RoboDK station: ESTACION KR10.rdk

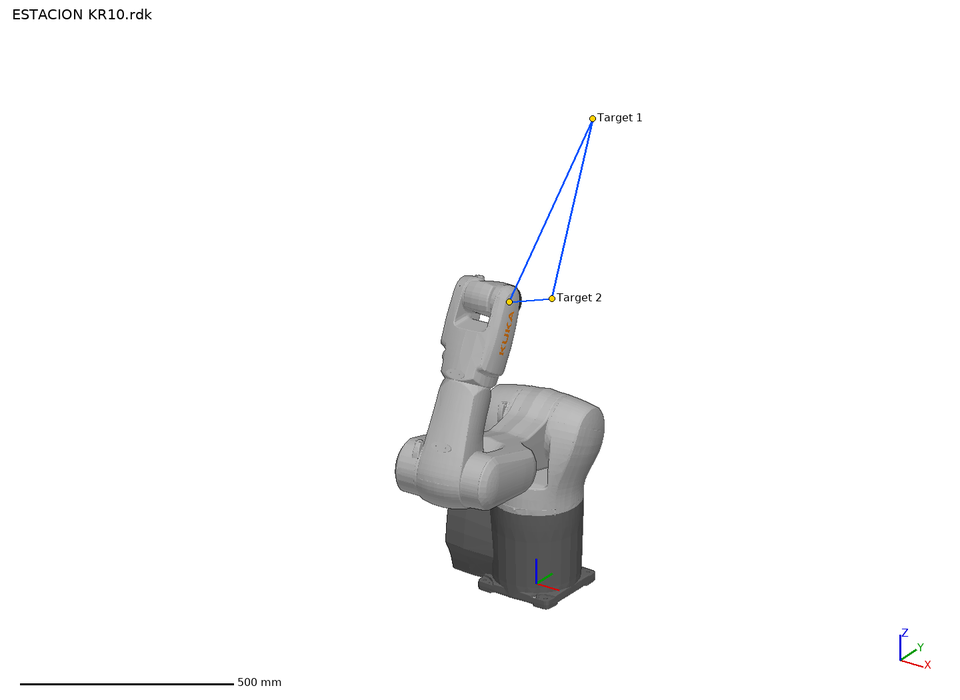
[picture v0: the station drawn from its stored meshes, robots at their saved joint values, targets as dots, program paths as lines]
Station ESTACION KR10 (saved by RoboDK 5.6.7). Poses are relative to the parent item; angles as X-Y-Z fixed-axis rotations.
  - frame KUKA KR 10 R900-2 Base at (0, 0, 0) mm
    - robot KUKA KR 10 R900-2: 6 axes, payload 10 kg, reach 901 mm, repeatability 0.03 mm, weight 52 kg
        modified DH rows (alpha deg, a mm, theta deg, d mm): 0, 0, 0, 400; -90, 25, 0, 0; 0, 455, -90, 0; -90, 25, 0, 420; 90, 0, 0, 0; -90, 0, 180, 90
        joint limits [-170, -190, -120, -185, -120, -350] to [170, 45, 156, 185, 120, 350]; home [0, -90, 90, 0, 0, 0]; saved at [-96.71, -171.34, 110.55, 9.97, 88.38, 69.15]
    - target Target 1 (Cartesian target) at (176.61, -22.09, 1268.28) mm, rotated rx 0 ry 16.57 rz -7.13 deg; joints [7.13, -104.931, 53.874, 0, -22.373, 0] of KUKA KR 10 R900-2
    - target Target 2 (Cartesian target) at (162.12, -169.54, 854.79) mm, rotated rx 176.4 ry 73.21 rz 172.77 deg; joints [65.15, -123.65, 113.03, -66.47, 66.83, 69.15] of KUKA KR 10 R900-2
    - target Target 3 (Cartesian target) at (34.52, -160.15, 806.28) mm, rotated rx -117.97 ry 13.68 rz -11.66 deg; joints [-96.71, -171.34, 110.55, 9.97, 88.38, 69.15] of KUKA KR 10 R900-2
  - program Prog1 (9 instructions, listed below)
  - Python program HandTrackingModule (listed below)
  - Python program FaceHandDetect (listed below)
  - Python program Prog2_vision (listed below)
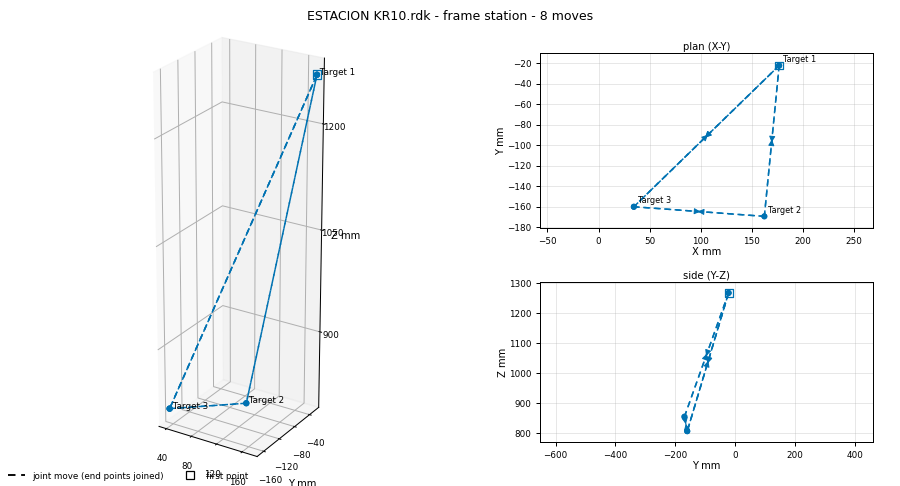
[picture p0: tool path of ESTACION KR10.rdk in frame station, 8 of 8 moves have a stored position in this frame; points joined in program order, loops and branches not executed]

--- program Prog1 (robot KUKA KR 10 R900-2) ---
  Est. Ref.: KUKA KR 10 R900-2 Base
  MoveJ (Target 1)
  MoveJ (Target 2)
  MoveJ (Target 3)
  MoveJ (Target 1)
  MoveJ (Target 3)
  MoveJ (Target 2)
  MoveJ (Target 1)
  MoveJ (Target 3)

--- Python program HandTrackingModule ---
import cv2 as cv
import mediapipe as mp
import time
import math
import numpy as np
import matplotlib.pyplot as plt

## EN PROGRESSO ###

class handDetector():
    def __init__(self,mode=False, maxHands=2,modelC=1,detectConf=0.5,trackConf=0.5):
        self.mode=mode
        self.maxHands=maxHands
        self.modelC = modelC
        self.detectConf=detectConf
        self.trackConf=trackConf

        self.mpHands = mp.solutions.hands
        self.hands = self.mpHands.Hands(self.mode,self.maxHands,self.modelC,self.detectConf,self.trackConf)
        self.mpDraw = mp.solutions.drawing_utils

        self.tipIds = [4, 8, 12, 16, 20]

    def findHands(self,img,draw=True):
        imgRGB=cv.cvtColor(img,cv.COLOR_BGR2RGB)
        nHands = 0
        self.results=self.hands.process(imgRGB)

        if self.results.multi_hand_landmarks:
            nHands = len(self.results.multi_hand_landmarks)
            for handLMs in self.results.multi_hand_landmarks:
                if draw:
                    self.mpDraw.draw_landmarks(img,handLMs,self.mpHands.HAND_CONNECTIONS)
        return img, nHands



    def findPos(self,img,handNumb=0,draw=False,palmLM = False, drawPalm = False):

        lmList = []
        if self.results.multi_hand_landmarks:
            myHand = self.results.multi_hand_landmarks[handNumb]
            for i,lm in enumerate(myHand.landmark):
                h,w,c=img.shape
                cx,cy,cz=int(lm.x*w),int(lm.y*h),lm.z
                lmList.append([i,cx,cy,cz])
                if draw:
                    cv.circle(img, (cx,cy), 5, (255,255,0), cv.FILLED)
            if palmLM:
                palmMarks = [0, 1, 5, 9, 13, 17]
                palmX, palmY, palmZ = 0, 0, 0
                for id in palmMarks:
                    palmX += lmList[id][1]
                    palmY += lmList[id][2]
                    palmZ += lmList[id][3]
                palm = [21, int(palmX/6), int(palmY/6), palmZ/6]
                lmList.append(palm)
                if drawPalm:
                    cv.circle(img, (palm[1],palm[2]), 5, (255,255,0), cv.FILLED)
        return lmList

    def lmDistance(self,lm1,lm2):
        dx = lm2[1]-lm1[1]
        dy = lm2[2]-lm1[2]
        dist = math.sqrt((dx**2)+(dy**2))
        return int(dist)

    def fingersState(self,lmList):
        fingersUp = []
        fingersCount = 0
        for id in self.tipIds:
            if id == 4:
                distP = self.lmDistance(lmList[id],lmList[17])
                distF = self.lmDistance(lmList[id-2],lmList[17])
            else:
                distP = self.lmDistance(lmList[id],lmList[0])
                distF = self.lmDistance(lmList[id-2],lmList[0])
            if distP > distF:
                fingersCount += 1
                fingersUp.append(1)
            else:
                fingersUp.append(0)
        return fingersUp, fingersCount



    def fingerVector(self, handNumb = 0, finger = 1):
        if self.results.multi_hand_landmarks and finger >= 0 and finger < 5:
            id = self.tipIds[finger]
            myHand = self.results.multi_hand_landmarks[handNumb]
            tipPos = myHand.landmark[id]
            basePos = myHand.landmark[id-2]
            x, y , z= (tipPos.x - basePos.x), (tipPos.y - basePos.y), (tipPos.z - basePos.z)
            mag = math.sqrt(x*x+y*y+z*z)
            vec = [x/mag,y/mag,z/mag]
            return vec
        else:
            return None


def main():
    cap = cv.VideoCapture(0)
    capW = int(cap.get(cv.CAP_PROP_FRAME_WIDTH))
    capH = int(cap.get(cv.CAP_PROP_FRAME_HEIGHT))
    pTime = 0
    cTime = 0

    detector=handDetector(maxHands= 1)

    fig = plt.figure()
    start =[0,0,0]


    x, y, z = int(capW/2), int(capH/2), 40
    pos = [x, y, z]
    vel = [0, 0, 0]

    while True:
        success , frame = cap.read()

        # gray = cv.cvtColor(frame,cv.COLOR_BGR2GRAY)
        # gFrame = cv.cvtColor(gray,cv.COLOR_GRAY2RGB)
        #cv.imshow('return to BGR',gFrame)
        frame = cv.flip(frame,1)
        frame, nHands = detector.findHands(frame)
        lmList = detector.findPos(frame,draw=True, palmLM = True, drawPalm = True)
        fingerVec= detector.fingerVector()
        #print('vector dedo:',fingerVec)
        cv.circle(frame,(pos[0],pos[1]),10,(0,0,255),-1)
        cv.putText(frame,'pos:'+str(pos),(20,80),cv.FONT_HERSHEY_COMPLEX,
         0.5,(0,255,0),thickness=1)
        cv.putText(frame,'vel:'+str(vel),(20,120),cv.FONT_HERSHEY_COMPLEX,
         0.5,(0,255,0),thickness=1)


        if len(lmList) != 0:
            print('palm pos:',10*lmList[21][3])
            fingerState,_ = detector.fingersState(lmList=lmList)
            cv.putText(frame,'fingerState:'+str(fingerState),(20,180),cv.FONT_HERSHEY_COMPLEX,
            0.5,(0,255,0),thickness=1)

            vel[0] = int(10*fingerVec[0])
            vel[1] = int(10*fingerVec[1])
            vel[2] = int(10*fingerVec[2])

            if fingerState == [0,1,0,0,0] or fingerState == [1,1,0,0,0]:
                pos[0] += vel[0]
                pos[1] += vel[1]
                pos[2] += vel[2]

        else:
            vel = [0,0,0]

        ax = plt.axes(projection = '3d')
        ax.set_xlim([-10,10])
        ax.set_ylim([-10,10])
        ax.set_zlim([-10,10])
        ax.quiver(start[0],start[1],start[2],vel[2],vel[0],-vel[1])
        ax.view_init(10,10)
        plt.pause(0.05) #Interrupcion de 0.05ms para poder visualizar los histogramas correctamente
        fig.clear()



        if pos[0]>capW:
            pos[0] = 0
        if pos[0]<0:
            pos[0] = capW
        if pos[1]>capH:
            pos[1] = 0
        if pos[1]<0:
            pos[1] = capH
        if pos[2]>80:
            pos[2] = 1
        if pos[2]<=0:
            pos[2] = 80







        cTime = time.time()
        fps = 1/(cTime-pTime)
        pTime = cTime
        cv.putText(frame,'fps:'+str(int(fps)),(20,40),cv.FONT_HERSHEY_COMPLEX,
         1,(0,255,0),thickness=2)

        cv.imshow('Video',frame)
        if cv.waitKey(20) & 0xFF==27:
            break

    cap.release()
    cv.destroyAllWindows()

if __name__=='__main__':
    main()

--- Python program FaceHandDetect ---
import cv2 as cv
import numpy as np
import os
import HandTrackingModule as htm
###################
path = 'haar_face.xml'
cameraN = 0
objectName = 'face'
frameWidth = 640
frameHeight = 480
####################

detector = htm.handDetector(detectConf=0.7)

capture= cv.VideoCapture(cameraN)
capture.set(3,frameWidth)
capture.set(4,frameHeight)

def empty(a):
    pass

#  CREATE TRACKBARS:
cv.namedWindow('display')
cv.resizeWindow('display',frameWidth,frameHeight+100)
cv.createTrackbar('Scale','display',400,1000,empty)
cv.createTrackbar('Neight','display',8,20,empty)
cv.createTrackbar('Min Area','display',0,100000,empty)

#  LOAD HAAR CASCADE CLASSIFIER:
cascade=cv.CascadeClassifier(path)

def cornerRect(img, bbox, l=30, t=5, rt=1,
               colorR=(255, 0, 255), colorC=(0, 255, 0)):
    """
    :param img: Image to draw on.
    :param bbox: Bounding box [x, y, w, h]
    :param l: length of the corner line
    :param t: thickness of the corner line
    :param rt: thickness of the rectangle
    :param colorR: Color of the Rectangle
    :param colorC: Color of the Corners
    :return:
    """
    x, y, w, h = bbox
    x1, y1 = x + w, y + h
    if rt != 0:
        cv.rectangle(img, bbox, colorR, rt)
    # Top Left  x,y
    cv.line(img, (x, y), (x + l, y), colorC, t)
    cv.line(img, (x, y), (x, y + l), colorC, t)
    # Top Right  x1,y
    cv.line(img, (x1, y), (x1 - l, y), colorC, t)
    cv.line(img, (x1, y), (x1, y + l), colorC, t)
    # Bottom Left  x,y1
    cv.line(img, (x, y1), (x + l, y1), colorC, t)
    cv.line(img, (x, y1), (x, y1 - l), colorC, t)
    # Bottom Right  x1,y1
    cv.line(img, (x1, y1), (x1 - l, y1), colorC, t)
    cv.line(img, (x1, y1), (x1, y1 - l), colorC, t)

    return img

while True:

    isTrueis,frame = capture.read()
    frame = cv.flip(frame,1)
    gray=cv.cvtColor(frame,cv.COLOR_BGR2GRAY)

    scaleVal = 1+(cv.getTrackbarPos('Scale','display')/1000)
    neig = cv.getTrackbarPos('Neight','display')

    objects=cascade.detectMultiScale(gray,scaleVal,neig)
    faceDetect = False
    safetyZone = None
    frame, nHands = detector.findHands(frame)
    lmList = detector.findPos(frame,draw=True, palmLM = True, drawPalm = True)
    for (x,y,w,h) in objects:
        area = w*h
        minArea = cv.getTrackbarPos('Min Area','display')
        if area > minArea:
            safetyZone = (int(x-1.3*w),y,w,h)
            cv.rectangle(frame,(x,y),(x+w,y+h),(0,255,0),thickness=2)
            cornerRect(frame, safetyZone, l=30, t=5, rt=1,colorR=(255, 0, 255), colorC=(0, 0, 255))
            cv.putText(frame, objectName, (x,y-5), cv.FONT_HERSHEY_COMPLEX_SMALL,
            1.0, (0,255,0), thickness=2)
            faces_roi=frame[y:y+h,x:x+w]
            faceDetect = True

    if faceDetect:
        lx , rx, uy, dy = safetyZone[0], safetyZone[0]+safetyZone[2], safetyZone[1], safetyZone[1]+safetyZone[3]
        if nHands > 0:
            px, py = lmList[21][1], lmList[21][2]

            if lx < px < rx and uy < py < dy:
                cornerRect(frame, safetyZone, l=30, t=5, rt=1,colorR=(255, 0, 255), colorC=(0, 255, 0))
                fingersState, fingerCount = detector.fingersState(lmList)
                fingersState.reverse()
                print(fingersState)
                # for i in fingersState:
                #     ylabel = int(frameHeight*0.8)


    cv.imshow('Video',frame)

    if cv.waitKey(20) & 0xFF==27:
        break

capture.release()
cv.destroyAllWindows()

--- Python program Prog2_vision ---
# Type help("robodk.robolink") or help("robodk.robomath") for more information
# Press F5 to run the script
# Documentation: https://robodk.com/doc/en/RoboDK-API.html
# Reference:     https://robodk.com/doc/en/PythonAPI/robodk.html
# Note: It is not required to keep a copy of this file, your Python script is saved with your RDK project
# Draw a hexagon around Target 1
from robolink import *    # RoboDK's API
from robodk import *      # Math toolbox for robots
import mediapipe as mp

# Start the RoboDK API:
RDK = Robolink()

# Get the robot (first robot found):
robot = RDK.Item('', ITEM_TYPE_ROBOT)

# Get the reference target by name:
target = RDK.Item('Target 1')
target2 = RDK.Item('Target 2')
target3 = RDK.Item('Target 3')
target_pose = target.Pose()
xyz_ref = target_pose.Pos()

# Move the robot to the reference point:
robot.MoveJ(target)
robot.MoveJ(target2)
robot.MoveJ(target3)

## Control por Visión ##
# El programa mueve el robot de uno de los targets definidos al otro en funcion de los dedos que se levanten(índice/índice+corazón)
import cv2 as cv
import mediapipe as mp
import time
import math


def findPos(img,results,handNumb=0,draw=False,palmLM = False, drawPalm = False):

    lmList = []
    if results.multi_hand_landmarks:
        myHand = results.multi_hand_landmarks[handNumb]
        for i,lm in enumerate(myHand.landmark):
            h,w,c=img.shape
            cx,cy,cz=int(lm.x*w),int(lm.y*h),lm.z
            lmList.append([i,cx,cy,cz])
            if draw:
                cv.circle(img, (cx,cy), 5, (255,255,0), cv.FILLED)
        if palmLM:
            palmMarks = [0, 1, 5, 9, 13, 17]
            palmX, palmY, palmZ = 0, 0, 0
            for id in palmMarks:
                palmX += lmList[id][1]
                palmY += lmList[id][2]
                palmZ += lmList[id][3]
            palm = [21, int(palmX/6), int(palmY/6), palmZ/6]
            lmList.append(palm)
            if drawPalm:
                cv.circle(img, (palm[1],palm[2]), 5, (255,255,0), cv.FILLED)
    return lmList

def lmDistance(lm1,lm2):
    dx = lm2[1]-lm1[1]
    dy = lm2[2]-lm1[2]
    dist = math.sqrt((dx**2)+(dy**2))
    return int(dist)

def fingersState(lmList):
    fingersUp = []
    fingersCount = 0
    tipIds = [4, 8, 12, 16, 20]
    for id in tipIds:
        if id == 4:
            distP = lmDistance(lmList[id],lmList[17])
            distF = lmDistance(lmList[id-2],lmList[17])
        else:
            distP = lmDistance(lmList[id],lmList[0])
            distF = lmDistance(lmList[id-2],lmList[0])
        if distP > distF:
            fingersCount += 1
            fingersUp.append(1)
        else:
            fingersUp.append(0)
    return fingersUp, fingersCount


cap = cv.VideoCapture(0)
mpHands = mp.solutions.hands
hands = mpHands.Hands()
mpDraw = mp.solutions.drawing_utils

pTime = 0
cTime = 0


while True:
    success , frame = cap.read()
    frame = cv.flip(frame,1)
    frameRGB=cv.cvtColor(frame,cv.COLOR_BGR2RGB)
    results=hands.process(frameRGB)
    lmList = findPos(frame,results,handNumb=0,draw=True,palmLM = False, drawPalm = False)
    if len(lmList) != 0:
        fingerState, fingersCount = fingersState(lmList)
        cv.putText(frame,'fingerState:'+str(fingerState),(20,100),cv.FONT_HERSHEY_COMPLEX,
                   0.5,(0,255,0),thickness=1)
        if fingerState == [0,1,0,0,0]:
            cv.putText(frame,'Target 1',(200,300),cv.FONT_HERSHEY_COMPLEX,
                   1,(0,0,255),thickness=1)
            robot.MoveJ(target)
            robot.RunInstruction('Program_Done')
        if fingerState == [0,1,1,0,0]:
            cv.putText(frame,'Target 2',(200,300),cv.FONT_HERSHEY_COMPLEX,
                   1,(0,0,255),thickness=1)
            robot.MoveJ(target2)
            robot.RunInstruction('Program_Done')
        if fingerState == [0,1,1,1,0]:
            cv.putText(frame,'Target 2',(200,300),cv.FONT_HERSHEY_COMPLEX,
                   1,(0,0,255),thickness=1)
            robot.MoveJ(target3)
            robot.RunInstruction('Program_Done')



    cTime = time.time()
    fps = 1/(cTime-pTime)
    pTime = cTime

    cv.putText(frame,'fps:'+str(int(fps)),(20,40),cv.FONT_HERSHEY_COMPLEX,
    1,(0,255,0),thickness=2)

    cv.imshow('Video',frame)
    if cv.waitKey(20) & 0xFF==27:
        break


cap.release()
cv.destroyAllWindows()

# Trigger a program call at the end of the movement
robot.RunInstruction('Program_Done')
